(* IEC 61131-3 sources: CS_4_Aufzugsteuerung/src/Stations/CP112/Steuerung/Class/clsTuerSensorik, 1 file *)

(* ---- clsTuerSensorik.st ---- *)
(*!
<Class
	Name               = "clsTuerSensorik"
	Revision           = "0.0"
	RealtimeTask       = "false"
	CyclicTask         = "true"
	DefCyclictime      = "1 ms"
	BackgroundTask     = "false"
	Sigmatek           = "false"
	OSInterface        = "false"
	HighPriority       = "false"
	Automatic          = "false"
	UpdateMode         = "Prescan"
	SharedCommandTable = "true"
	Objectsize         = "(284,120)">
	<Channels>
		<Server Name="ClassSvr" Visualized="false" Initialize="false" WriteProtected="true" Retentive="false"/>
		<Server Name="sVisuTuer" Visualized="true" Initialize="false" WriteProtected="false" Retentive="false"/>
		<Client Name="cFahrzeit" Required="false" Internal="false"/>
		<Client Name="cTimer" Required="true" Internal="false"/>
	</Channels>
</Class>
*)
clsTuerSensorik : CLASS
	TYPE
	  Tuerstates : DINT;
	END_TYPE
  //Servers:
	ClassSvr 	: SvrChCmd_DINT;
	sVisuTuer 	: SvrCh_DINT;
  //Clients:
	cTimer 	: CltChCmd_clsTimer;
	cFahrzeit 	: CltCh_UDINT;
  //Variables:
		xAuf 	: BOOL;
		xZu 	: BOOL;
  //Functions:

	FUNCTION VIRTUAL GLOBAL CyWork
		VAR_INPUT
			EAX 	: UDINT;
		END_VAR
		VAR_OUTPUT
			state (EAX) 	: UDINT;
		END_VAR;

	FUNCTION GLOBAL zu;

	FUNCTION GLOBAL auf;

	FUNCTION GLOBAL istzu
		VAR_OUTPUT
			xOut 	: BOOL;
		END_VAR;

	FUNCTION GLOBAL istauf
		VAR_OUTPUT
			xOut 	: BOOL;
		END_VAR;
  //Tables:
	FUNCTION @STD
		VAR_OUTPUT
			ret_code	: CONFSTATES;
		END_VAR;
	FUNCTION GLOBAL TAB @CT_;
END_CLASS;

#pragma usingLtd clsTimer

FUNCTION VIRTUAL GLOBAL clsTuerSensorik::CyWork
	VAR_INPUT
		EAX 	: UDINT;
	END_VAR
	VAR_OUTPUT
		state (EAX) 	: UDINT;
	END_VAR

  cFahrzeit := cFahrzeit.Read();

  //Uebergabe an HMI
  sVisuTuer := xAuf;

	state := READY;

END_FUNCTION

FUNCTION GLOBAL clsTuerSensorik::zu

  //pruefen ob schon zu
  IF NOT xZu AND NOT cTimer.running() THEN
     cTimer.Start(_time := cFahrzeit);
  END_IF;

  IF cTimer.elapsed() THEN
      xAuf := FALSE;
      xZu := TRUE;
  END_IF;

END_FUNCTION

FUNCTION GLOBAL clsTuerSensorik::auf

  // Pruefen ob schon offen
  IF NOT xAuf AND NOT cTimer.running()  THEN
    cTimer.Start(_time := cFahrzeit);
  END_IF;

  IF cTimer.elapsed() THEN
      xAuf := TRUE;
      xZu := FALSE;
  END_IF;

END_FUNCTION

FUNCTION GLOBAL clsTuerSensorik::istzu
	VAR_OUTPUT
		xOut 	: BOOL;
	END_VAR
 xOut := xZu;
END_FUNCTION

FUNCTION GLOBAL clsTuerSensorik::istauf
	VAR_OUTPUT
		xOut 	: BOOL;
	END_VAR
 xOut := xAuf;
END_FUNCTION
